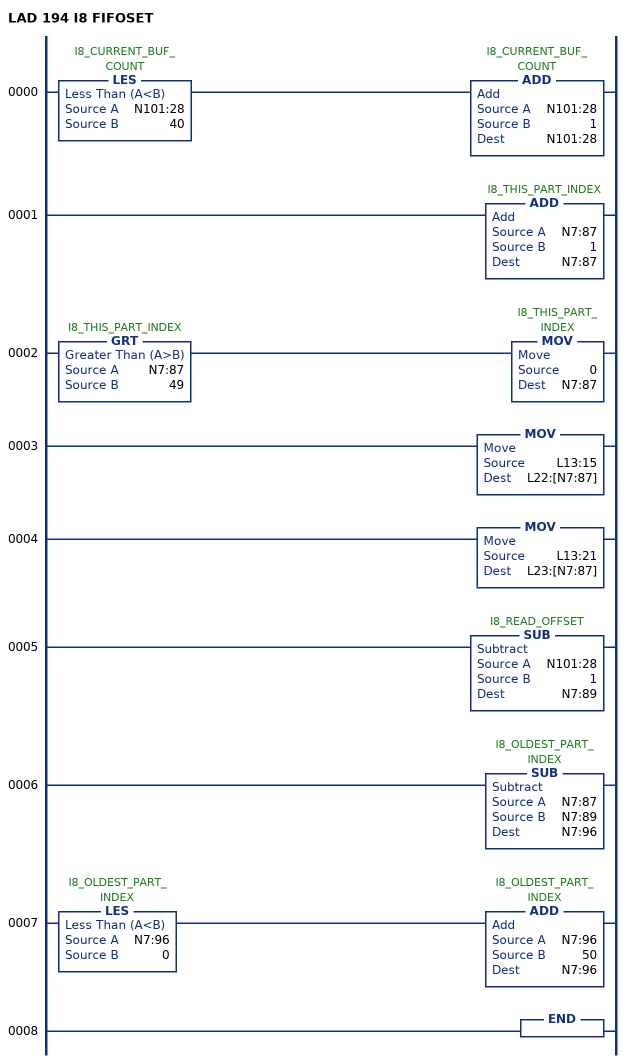
% Rung: 0 %
SOR LES N101:28 40 ADD N101:28 1 N101:28 EOR
%   N101:28  I8_CURRENT_BUF_COUNT %
% Rung: 1 %
SOR ADD N7:87 1 N7:87 EOR
%   N7:87  I8_THIS_PART_INDEX %
% Rung: 2 %
SOR GRT N7:87 49 MOV 0 N7:87 EOR
%   N7:87  I8_THIS_PART_INDEX %
% Rung: 3 %
SOR MOV L13:15 L22:[N7:87] EOR
%   L13:15  THE_TIME %
%   N7:87  I8_THIS_PART_INDEX %
% Rung: 4 %
SOR MOV L13:21 L23:[N7:87] EOR
%   L13:21  TOP_POSITION %
%   N7:87  I8_THIS_PART_INDEX %
% Rung: 5 %
SOR SUB N101:28 1 N7:89 EOR
%   N101:28  I8_CURRENT_BUF_COUNT %
%   N7:89  I8_READ_OFFSET %
% Rung: 6 %
SOR SUB N7:87 N7:89 N7:96 EOR
%   N7:87  I8_THIS_PART_INDEX %
%   N7:89  I8_READ_OFFSET %
%   N7:96  I8_OLDEST_PART_INDEX %
% Rung: 7 %
SOR LES N7:96 0 ADD N7:96 50 N7:96 EOR
%   N7:96  I8_OLDEST_PART_INDEX %
% Rung: 8 %
SOR END EOR

LADDER 195 "I8 FIFOGET"
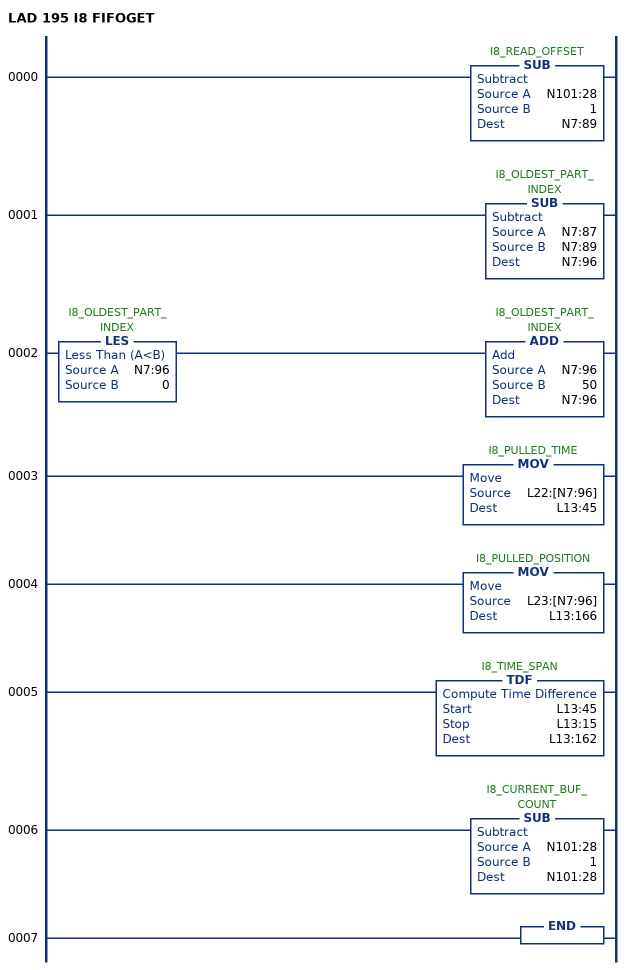
% Rung: 0 %
SOR SUB N101:28 1 N7:89 EOR
%   N101:28  I8_CURRENT_BUF_COUNT %
%   N7:89  I8_READ_OFFSET %
% Rung: 1 %
SOR SUB N7:87 N7:89 N7:96 EOR
%   N7:87  I8_THIS_PART_INDEX %
%   N7:89  I8_READ_OFFSET %
%   N7:96  I8_OLDEST_PART_INDEX %
% Rung: 2 %
SOR LES N7:96 0 ADD N7:96 50 N7:96 EOR
%   N7:96  I8_OLDEST_PART_INDEX %
% Rung: 3 %
SOR MOV L22:[N7:96] L13:45 EOR
%   N7:96  I8_OLDEST_PART_INDEX %
%   L13:45  I8_PULLED_TIME %
% Rung: 4 %
SOR MOV L23:[N7:96] L13:166 EOR
%   N7:96  I8_OLDEST_PART_INDEX %
%   L13:166  I8_PULLED_POSITION %
% Rung: 5 %
SOR TDF L13:45 L13:15 L13:162 EOR
%   L13:45  I8_PULLED_TIME %
%   L13:15  THE_TIME %
%   L13:162  I8_TIME_SPAN %
% Rung: 6 %
SOR SUB N101:28 1 N101:28 EOR
%   N101:28  I8_CURRENT_BUF_COUNT %
% Rung: 7 %
SOR END EOR

LADDER 196 "I8 DATA"
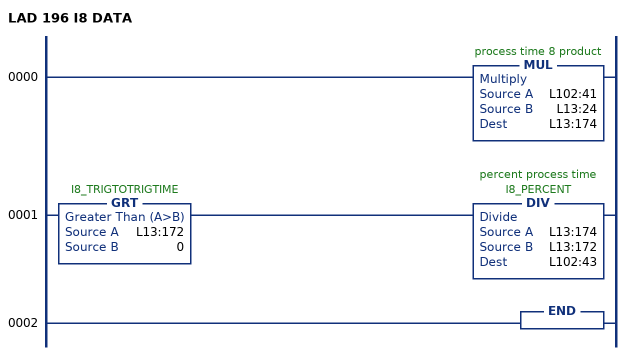
% Rung: 0 %
SOR MUL L102:41 L13:24 L13:174 EOR
%   L102:41  I8_PROCESSTIME %
%   L13:24  "multiplyer to make devision come out to a percentage" %
%   L13:174  "process time 8 product" %
% Rung: 1 %
SOR GRT L13:172 0 DIV L13:174 L13:172 L102:43 EOR
%   L13:172  I8_TRIGTOTRIGTIME %
%   L13:174  "process time 8 product" %
%   L102:43  I8_PERCENT  "percent process time" %
% Rung: 2 %
SOR END EOR

LADDER 197 "I8 FAULT"
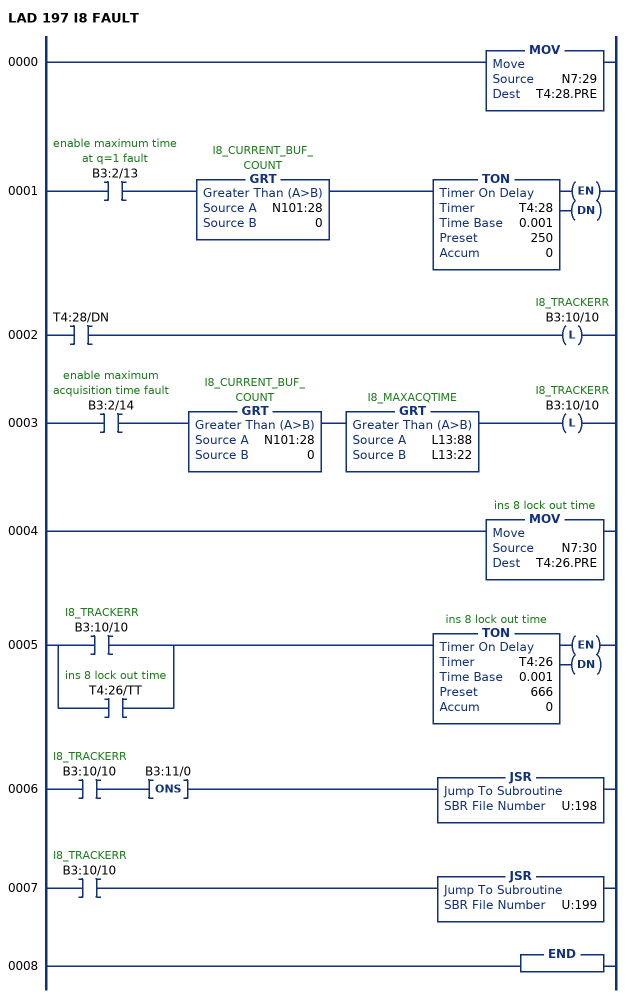
% Rung: 0 %
SOR MOV N7:29 T4:28.PRE EOR
%   N7:29  "max allowed ms time for q to be above 1 if safe fault is used" %
% Rung: 1 %
SOR XIC B3:2/13 GRT N101:28 0 TON T4:28 0.001 250 0 EOR
%   B3:2/13  "enable maximum time at q=1 fault" %
%   N101:28  I8_CURRENT_BUF_COUNT %
% Rung: 2 %
SOR XIC T4:28/DN OTL B3:10/10 EOR
%   B3:10/10  I8_TRACKERR %
% Rung: 3 %
SOR XIC B3:2/14 GRT N101:28 0 GRT L13:88 L13:22 OTL B3:10/10 EOR
%   B3:2/14  "enable maximum acquisition time fault" %
%   N101:28  I8_CURRENT_BUF_COUNT %
%   L13:88  I8_MAXACQTIME %
%   L13:22  "maximum of the longest acquire time allowed if maximum acquire time fault is enabled" %
%   B3:10/10  I8_TRACKERR %
% Rung: 4 %
SOR MOV N7:30 T4:26.PRE EOR
%   N7:30  "ms time setting to lock out inspection to give all pending images a chance to clear" %
%   T4:26  "ins 8 lock out time" %
% Rung: 5 %
SOR BST XIC B3:10/10 NXB XIC T4:26/TT BND TON T4:26 0.001 666 0 EOR
%   B3:10/10  I8_TRACKERR %
%   T4:26  "ins 8 lock out time" %
% Rung: 6 %
SOR XIC B3:10/10 ONS B3:11/0 JSR U:198 EOR
%   B3:10/10  I8_TRACKERR %
% Rung: 7 %
SOR XIC B3:10/10 JSR U:199 EOR
%   B3:10/10  I8_TRACKERR %
% Rung: 8 %
SOR END EOR

LADDER 198 "I8 FIX1"
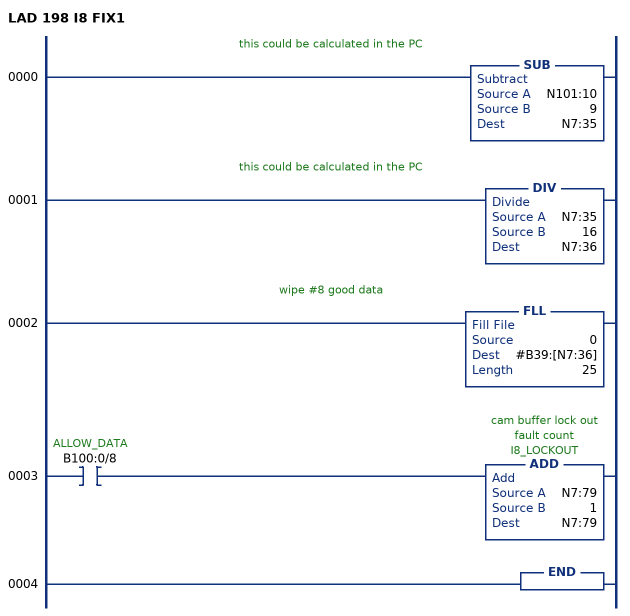
% Rung: 0 %
% this could be calculated in the PC %
SOR SUB N101:10 9 N7:35 EOR
%   N101:10  I8_TRIG_LOC %
% Rung: 1 %
% this could be calculated in the PC %
SOR DIV N7:35 16 N7:36 EOR
% Rung: 2 %
% wipe #8 good data %
SOR FLL 0 #B39:[N7:36] 25 EOR
% Rung: 3 %
SOR XIC B100:0/8 ADD N7:79 1 N7:79 EOR
%   B100:0/8  ALLOW_DATA %
%   N7:79  I8_LOCKOUT  "cam buffer lock out fault count" %
% Rung: 4 %
SOR END EOR

LADDER 199 "I8 FIX2"
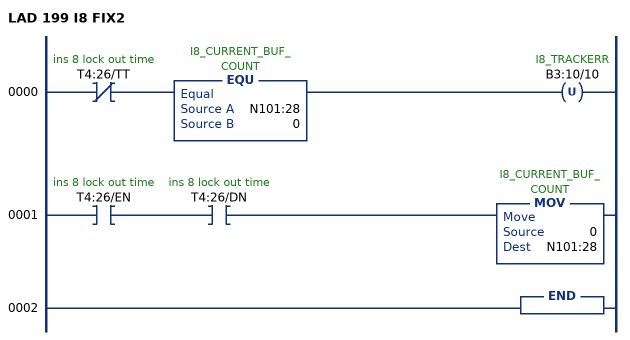
% Rung: 0 %
SOR XIO T4:26/TT EQU N101:28 0 OTU B3:10/10 EOR
%   T4:26  "ins 8 lock out time" %
%   N101:28  I8_CURRENT_BUF_COUNT %
%   B3:10/10  I8_TRACKERR %
% Rung: 1 %
SOR XIC T4:26/EN XIC T4:26/DN MOV 0 N101:28 EOR
%   T4:26  "ins 8 lock out time" %
%   N101:28  I8_CURRENT_BUF_COUNT %
% Rung: 2 %
SOR END EOR

LADDER 200 "PASS BLOW"
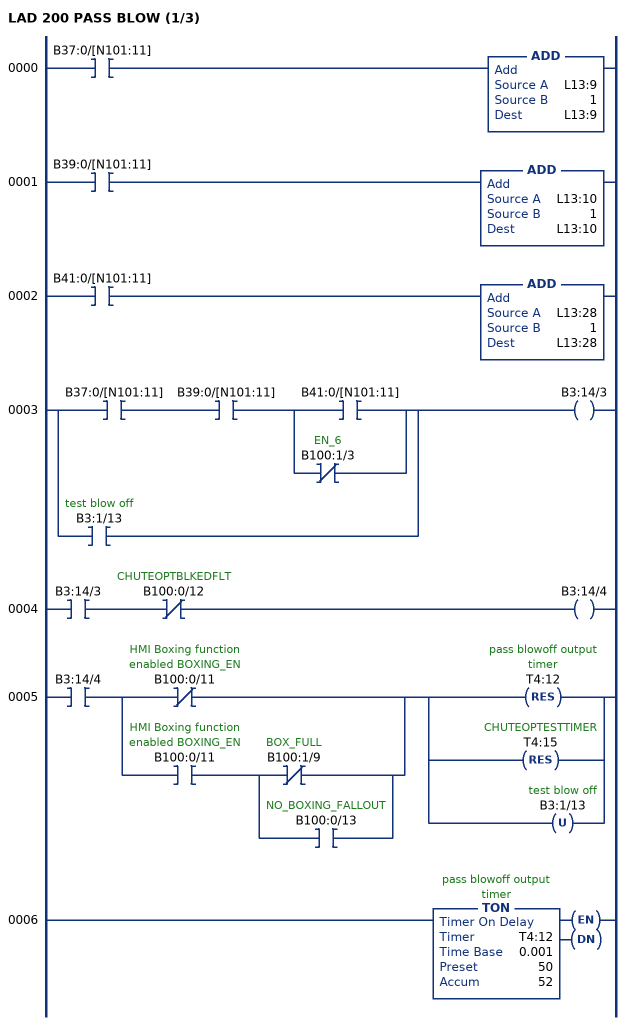
% Rung: 0 %
SOR XIC B37:0/[N101:11] ADD L13:9 1 L13:9 EOR
%   B37:0  TOP_OK_1 %
%   N101:11  BLOW_PT %
% Rung: 1 %
SOR XIC B39:0/[N101:11] ADD L13:10 1 L13:10 EOR
%   B39:0  TOP_OK_2 %
%   N101:11  BLOW_PT %
% Rung: 2 %
SOR XIC B41:0/[N101:11] ADD L13:28 1 L13:28 EOR
%   B41:0  TOP_OK_3 %
%   N101:11  BLOW_PT %
% Rung: 3 %
SOR BST XIC B37:0/[N101:11] XIC B39:0/[N101:11] BST XIC B41:0/[N101:11] NXB XIO B100:1/3 BND NXB XIC B3:1/13 BND OTE B3:14/3 EOR
%   B37:0  TOP_OK_1 %
%   N101:11  BLOW_PT %
%   B39:0  TOP_OK_2 %
%   B41:0  TOP_OK_3 %
%   B100:1/3  EN_6 %
%   B3:1/13  "test blow off" %
% Rung: 4 %
SOR XIC B3:14/3 XIO B100:0/12 OTE B3:14/4 EOR
%   B100:0/12  CHUTEOPTBLKEDFLT %
% Rung: 5 %
SOR XIC B3:14/4 BST XIO B100:0/11 NXB XIC B100:0/11 BST XIO B100:1/9 NXB XIC B100:0/13 BND BND BST RES T4:12 NXB RES T4:15 NXB OTU B3:1/13 BND EOR
%   B100:0/11  BOXING_EN  "HMI Boxing function enabled" %
%   B100:1/9  BOX_FULL %
%   B100:0/13  NO_BOXING_FALLOUT %
%   T4:12  "pass blowoff output timer" %
%   T4:15  CHUTEOPTESTTIMER %
%   B3:1/13  "test blow off" %
% Rung: 6 %
SOR TON T4:12 0.001 50 52 EOR
%   T4:12  "pass blowoff output timer" %

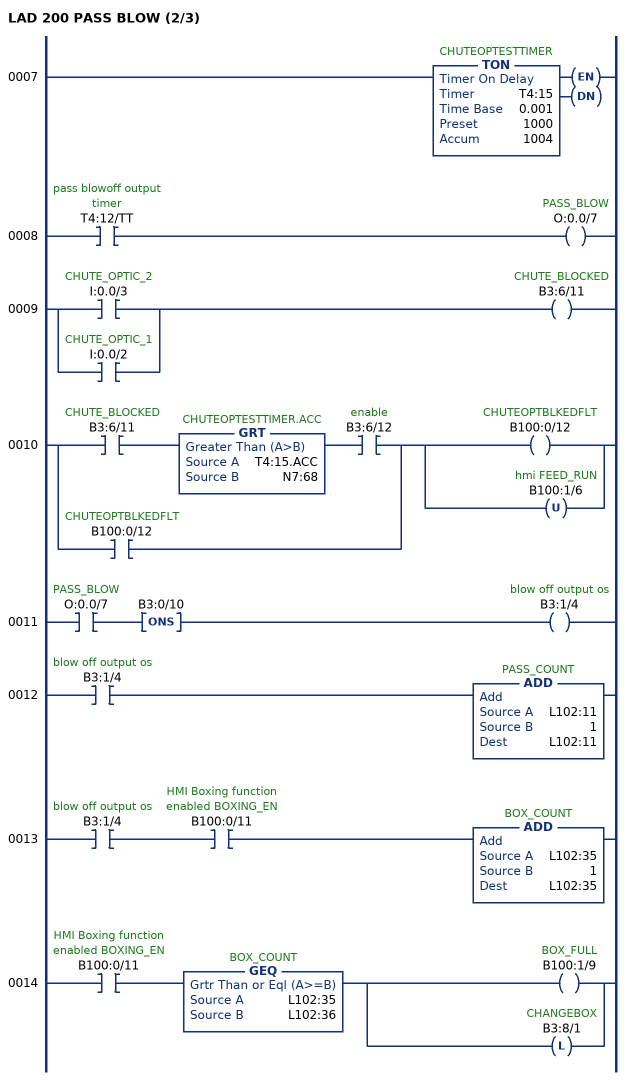
% Rung: 7 %
SOR TON T4:15 0.001 1000 1004 EOR
%   T4:15  CHUTEOPTESTTIMER %
% Rung: 8 %
SOR XIC T4:12/TT OTE O:0.0/7 EOR
%   T4:12  "pass blowoff output timer" %
%   O:0.0/7  PASS_BLOW %
% Rung: 9 %
SOR BST XIC I:0.0/3 NXB XIC I:0.0/2 BND OTE B3:6/11 EOR
%   I:0.0/3  CHUTE_OPTIC_2 %
%   I:0.0/2  CHUTE_OPTIC_1 %
%   B3:6/11  CHUTE_BLOCKED %
% Rung: 10 %
SOR BST XIC B3:6/11 GRT T4:15.ACC N7:68 XIC B3:6/12 NXB XIC B100:0/12 BND BST OTE B100:0/12 NXB OTU B100:1/6 BND EOR
%   B3:6/11  CHUTE_BLOCKED %
%   T4:15  CHUTEOPTESTTIMER %
%   B3:6/12  "enable" %
%   B100:0/12  CHUTEOPTBLKEDFLT %
%   B100:1/6  FEED_RUN  "hmi" %
% Rung: 11 %
SOR XIC O:0.0/7 ONS B3:0/10 OTE B3:1/4 EOR
%   O:0.0/7  PASS_BLOW %
%   B3:1/4  "blow off output os" %
% Rung: 12 %
SOR XIC B3:1/4 ADD L102:11 1 L102:11 EOR
%   B3:1/4  "blow off output os" %
%   L102:11  PASS_COUNT %
% Rung: 13 %
SOR XIC B3:1/4 XIC B100:0/11 ADD L102:35 1 L102:35 EOR
%   B3:1/4  "blow off output os" %
%   B100:0/11  BOXING_EN  "HMI Boxing function enabled" %
%   L102:35  BOX_COUNT %
% Rung: 14 %
SOR XIC B100:0/11 GEQ L102:35 L102:36 BST OTE B100:1/9 NXB OTL B3:8/1 BND EOR
%   B100:0/11  BOXING_EN  "HMI Boxing function enabled" %
%   L102:35  BOX_COUNT %
%   L102:36  BOX_LIMIT  "box count setpoint" %
%   B100:1/9  BOX_FULL %
%   B3:8/1  CHANGEBOX %

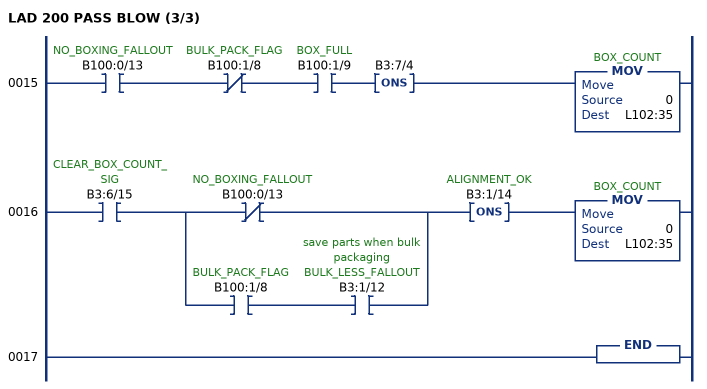
% Rung: 15 %
SOR XIC B100:0/13 XIO B100:1/8 XIC B100:1/9 ONS B3:7/4 MOV 0 L102:35 EOR
%   B100:0/13  NO_BOXING_FALLOUT %
%   B100:1/8  BULK_PACK_FLAG %
%   B100:1/9  BOX_FULL %
%   L102:35  BOX_COUNT %
% Rung: 16 %
SOR XIC B3:6/15 BST XIO B100:0/13 NXB XIC B100:1/8 XIC B3:1/12 BND ONS B3:1/14 MOV 0 L102:35 EOR
%   B3:6/15  CLEAR_BOX_COUNT_SIG %
%   B100:0/13  NO_BOXING_FALLOUT %
%   B100:1/8  BULK_PACK_FLAG %
%   B3:1/12  BULK_LESS_FALLOUT  "save parts when bulk packaging" %
%   B3:1/14  ALIGNMENT_OK %
%   L102:35  BOX_COUNT %
% Rung: 17 %
SOR END EOR

LADDER 235 "TESTTRIGS"    % highspeed test triggers, not necessary %
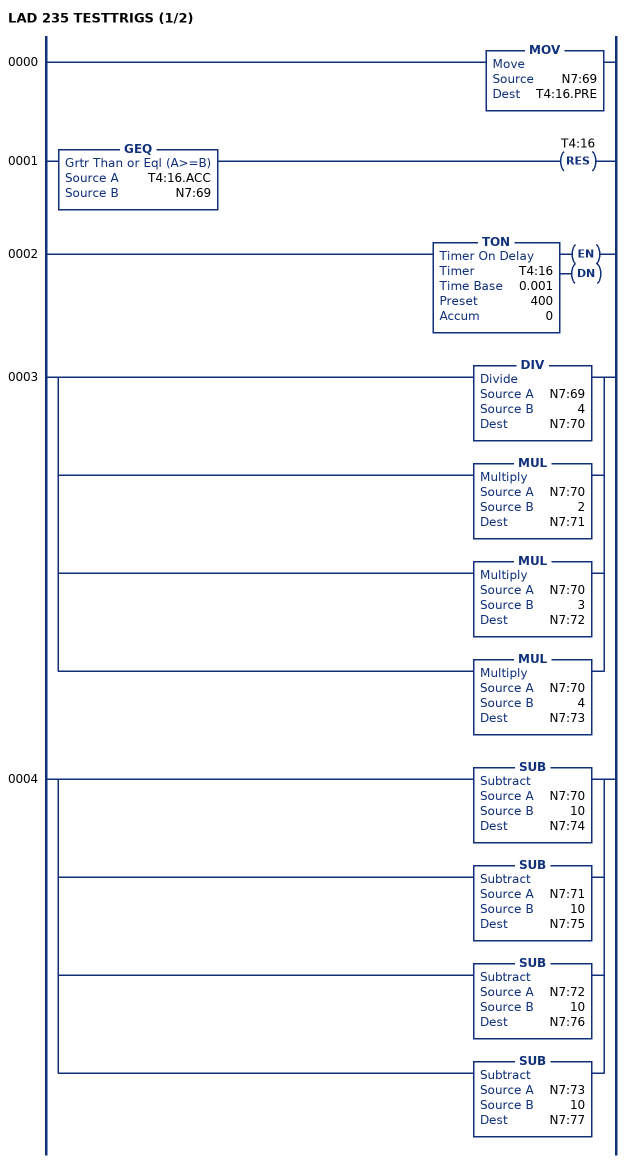
% Rung: 0 %
SOR MOV N7:69 T4:16.PRE EOR
% Rung: 1 %
SOR GEQ T4:16.ACC N7:69 RES T4:16 EOR
% Rung: 2 %
SOR TON T4:16 0.001 400 0 EOR
% Rung: 3 %
SOR BST DIV N7:69 4 N7:70 NXB MUL N7:70 2 N7:71 NXB MUL N7:70 3 N7:72 NXB MUL N7:70 4 N7:73 BND EOR
% Rung: 4 %
SOR BST SUB N7:70 10 N7:74 NXB SUB N7:71 10 N7:75 NXB SUB N7:72 10 N7:76 NXB SUB N7:73 10 N7:77 BND EOR

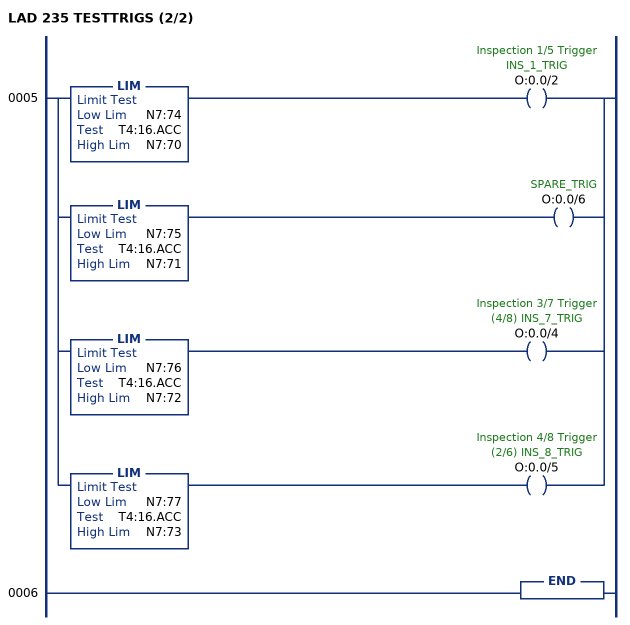
% Rung: 5 %
SOR BST LIM N7:74 T4:16.ACC N7:70 OTE O:0.0/2 NXB LIM N7:75 T4:16.ACC N7:71 OTE O:0.0/6 NXB LIM N7:76 T4:16.ACC N7:72 OTE O:0.0/4 NXB LIM N7:77 T4:16.ACC N7:73 OTE O:0.0/5 BND EOR
%   O:0.0/2  INS_1_TRIG  "Inspection 1/5 Trigger" %
%   O:0.0/6  SPARE_TRIG %
%   O:0.0/4  INS_7_TRIG  "Inspection 3/7 Trigger (4/8)" %
%   O:0.0/5  INS_8_TRIG  "Inspection 4/8 Trigger (2/6)" %
% Rung: 6 %
SOR END EOR

LADDER 236 "TESTTRIG1"
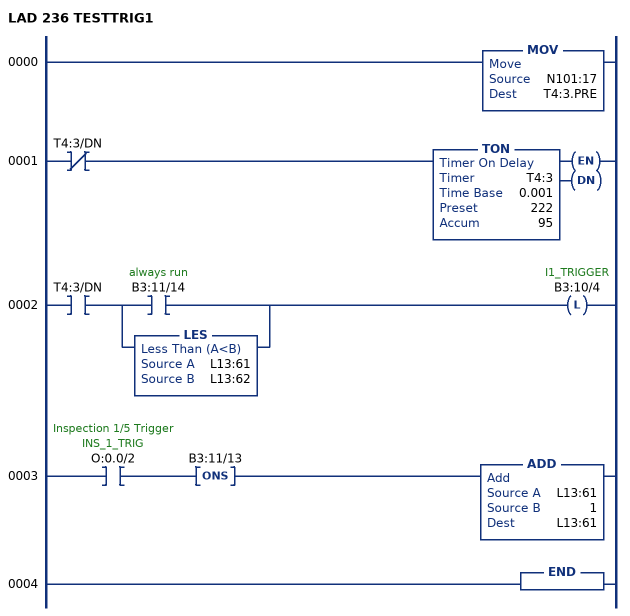
% Rung: 0 %
SOR MOV N101:17 T4:3.PRE EOR
%   N101:17  I1_TRIGTIME  "test trigger 1 interval" %
% Rung: 1 %
SOR XIO T4:3/DN TON T4:3 0.001 222 95 EOR
% Rung: 2 %
SOR XIC T4:3/DN BST XIC B3:11/14 NXB LES L13:61 L13:62 BND OTL B3:10/4 EOR
%   B3:11/14  "always run" %
%   B3:10/4  I1_TRIGGER %
% Rung: 3 %
SOR XIC O:0.0/2 ONS B3:11/13 ADD L13:61 1 L13:61 EOR
%   O:0.0/2  INS_1_TRIG  "Inspection 1/5 Trigger" %
% Rung: 4 %
SOR END EOR

LADDER 237 "TESTTRIG2"
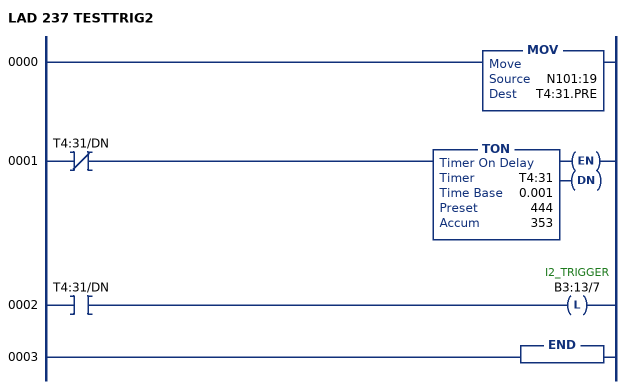
% Rung: 0 %
SOR MOV N101:19 T4:31.PRE EOR
%   N101:19  I2_I6_TRIGTIME  "test trgiger 2/6 interval" %
% Rung: 1 %
SOR XIO T4:31/DN TON T4:31 0.001 444 353 EOR
% Rung: 2 %
SOR XIC T4:31/DN OTL B3:13/7 EOR
%   B3:13/7  I2_TRIGGER %
% Rung: 3 %
SOR END EOR

LADDER 238 "TESTTRIG3"
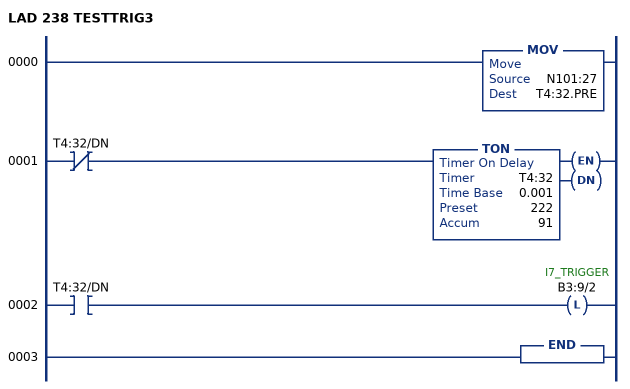
% Rung: 0 %
SOR MOV N101:27 T4:32.PRE EOR
%   N101:27  I7_TRIGTIME %
% Rung: 1 %
SOR XIO T4:32/DN TON T4:32 0.001 222 91 EOR
% Rung: 2 %
SOR XIC T4:32/DN OTL B3:9/2 EOR
%   B3:9/2  I7_TRIGGER %
% Rung: 3 %
SOR END EOR

LADDER 239 "TESTTRIG4"
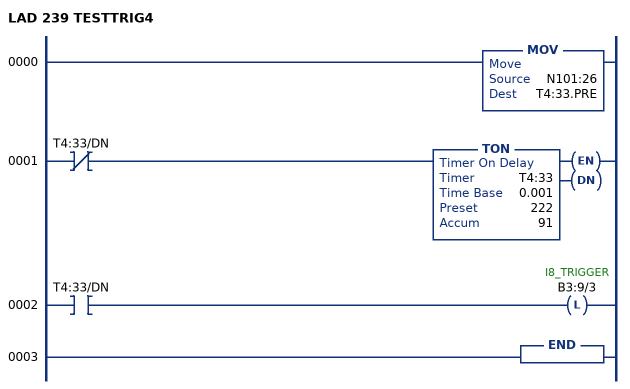
% Rung: 0 %
SOR MOV N101:26 T4:33.PRE EOR
%   N101:26  I8_TRIGTIME %
% Rung: 1 %
SOR XIO T4:33/DN TON T4:33 0.001 222 91 EOR
% Rung: 2 %
SOR XIC T4:33/DN OTL B3:9/3 EOR
%   B3:9/3  I8_TRIGGER %
% Rung: 3 %
SOR END EOR

LADDER 240 "TESTTRIG5"
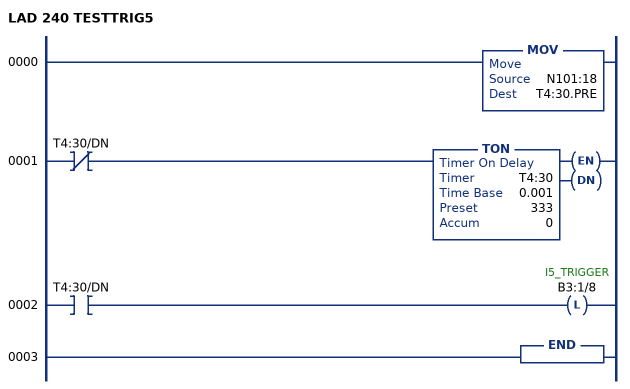
% Rung: 0 %
SOR MOV N101:18 T4:30.PRE EOR
%   N101:18  I5_TRIGTIME  "test trigger 5 interval" %
% Rung: 1 %
SOR XIO T4:30/DN TON T4:30 0.001 333 0 EOR
% Rung: 2 %
SOR XIC T4:30/DN OTL B3:1/8 EOR
%   B3:1/8  I5_TRIGGER %
% Rung: 3 %
SOR END EOR

LADDER 241 "TESTTRIG6"
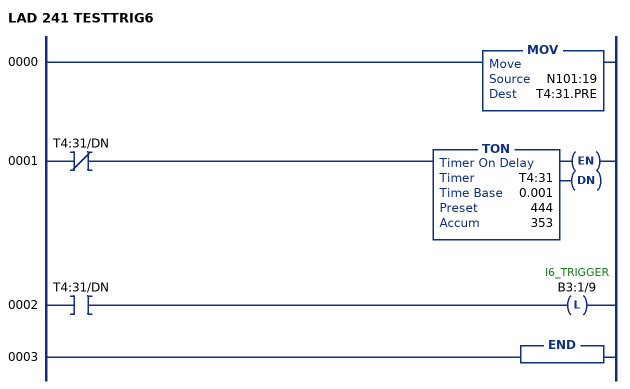
% Rung: 0 %
SOR MOV N101:19 T4:31.PRE EOR
%   N101:19  I2_I6_TRIGTIME  "test trgiger 2/6 interval" %
% Rung: 1 %
SOR XIO T4:31/DN TON T4:31 0.001 444 353 EOR
% Rung: 2 %
SOR XIC T4:31/DN OTL B3:1/9 EOR
%   B3:1/9  I6_TRIGGER %
% Rung: 3 %
SOR END EOR

LADDER 242 "TESTTRIG7"
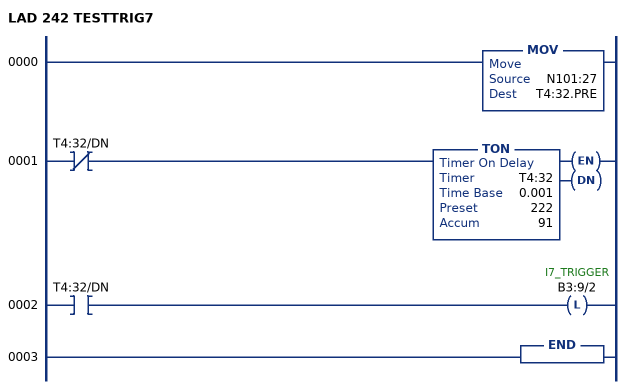
% Rung: 0 %
SOR MOV N101:27 T4:32.PRE EOR
%   N101:27  I7_TRIGTIME %
% Rung: 1 %
SOR XIO T4:32/DN TON T4:32 0.001 222 91 EOR
% Rung: 2 %
SOR XIC T4:32/DN OTL B3:9/2 EOR
%   B3:9/2  I7_TRIGGER %
% Rung: 3 %
SOR END EOR

LADDER 243 "TESTTRIG8"
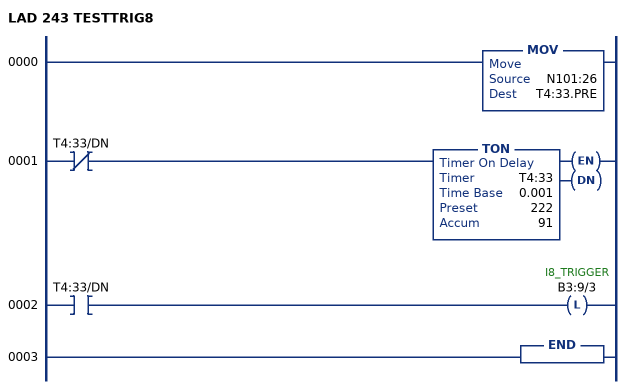
% Rung: 0 %
SOR MOV N101:26 T4:33.PRE EOR
%   N101:26  I8_TRIGTIME %
% Rung: 1 %
SOR XIO T4:33/DN TON T4:33 0.001 222 91 EOR
% Rung: 2 %
SOR XIC T4:33/DN OTL B3:9/3 EOR
%   B3:9/3  I8_TRIGGER %
% Rung: 3 %
SOR END EOR

LADDER 244 "PACKAGER"    % normal %
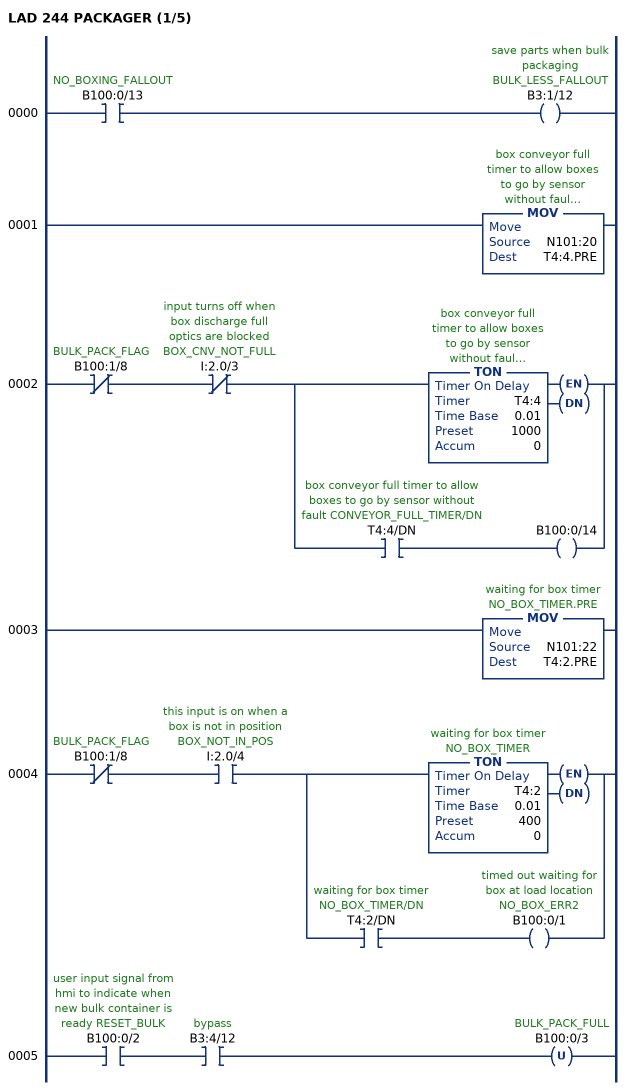
% Rung: 0 %
SOR XIC B100:0/13 OTE B3:1/12 EOR
%   B100:0/13  NO_BOXING_FALLOUT %
%   B3:1/12  BULK_LESS_FALLOUT  "save parts when bulk packaging" %
% Rung: 1 %
SOR MOV N101:20 T4:4.PRE EOR
%   N101:20  CONV_FULL_TIME_LIMIT  "time to allow box to pass box conveyor full sensor without fault" %
%   T4:4  CONVEYOR_FULL_TIMER  "box conveyor full timer to allow boxes to go by sensor without fault" %
% Rung: 2 %
SOR XIO B100:1/8 XIO I:2.0/3 BST TON T4:4 0.01 1000 0 NXB XIC T4:4/DN OTE B100:0/14 BND EOR
%   B100:1/8  BULK_PACK_FLAG %
%   I:2.0/3  BOX_CNV_NOT_FULL  "input turns off when box discharge full optics are blocked" %
%   T4:4  CONVEYOR_FULL_TIMER  "box conveyor full timer to allow boxes to go by sensor without fault" %
% Rung: 3 %
SOR MOV N101:22 T4:2.PRE EOR
%   N101:22  BOX_WAIT_TIME_LIMIT  "the time until waiting for box message in hmi (fault)" %
%   T4:2  NO_BOX_TIMER  "waiting for box timer" %
% Rung: 4 %
SOR XIO B100:1/8 XIC I:2.0/4 BST TON T4:2 0.01 400 0 NXB XIC T4:2/DN OTE B100:0/1 BND EOR
%   B100:1/8  BULK_PACK_FLAG %
%   I:2.0/4  BOX_NOT_IN_POS  "this input is on when a box is not in position" %
%   T4:2  NO_BOX_TIMER  "waiting for box timer" %
%   B100:0/1  NO_BOX_ERR2  "timed out waiting for box at load location" %
% Rung: 5 %
SOR XIC B100:0/2 XIC B3:4/12 OTU B100:0/3 EOR
%   B100:0/2  RESET_BULK  "user input signal from hmi to indicate when new bulk container is ready" %
%   B3:4/12  "bypass" %
%   B100:0/3  BULK_PACK_FULL %

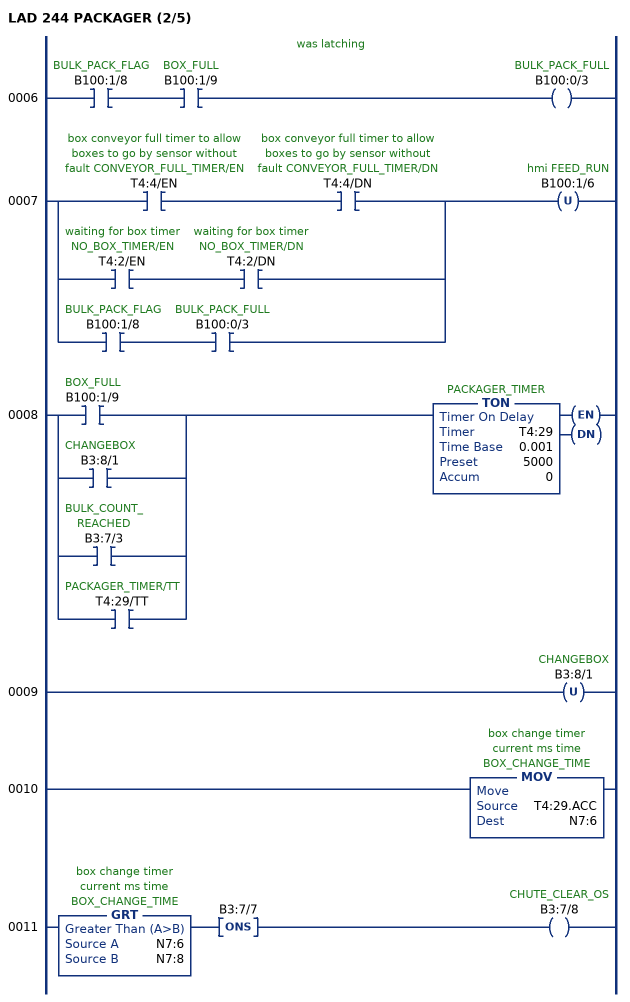
% Rung: 6 %
% was latching %
SOR XIC B100:1/8 XIC B100:1/9 OTE B100:0/3 EOR
%   B100:1/8  BULK_PACK_FLAG %
%   B100:1/9  BOX_FULL %
%   B100:0/3  BULK_PACK_FULL %
% Rung: 7 %
SOR BST XIC T4:4/EN XIC T4:4/DN NXB XIC T4:2/EN XIC T4:2/DN NXB XIC B100:1/8 XIC B100:0/3 BND OTU B100:1/6 EOR
%   T4:4  CONVEYOR_FULL_TIMER  "box conveyor full timer to allow boxes to go by sensor without fault" %
%   T4:2  NO_BOX_TIMER  "waiting for box timer" %
%   B100:1/8  BULK_PACK_FLAG %
%   B100:0/3  BULK_PACK_FULL %
%   B100:1/6  FEED_RUN  "hmi" %
% Rung: 8 %
SOR BST XIC B100:1/9 NXB XIC B3:8/1 NXB XIC B3:7/3 NXB XIC T4:29/TT BND TON T4:29 0.001 5000 0 EOR
%   B100:1/9  BOX_FULL %
%   B3:8/1  CHANGEBOX %
%   B3:7/3  BULK_COUNT_REACHED %
%   T4:29  PACKAGER_TIMER %
% Rung: 9 %
SOR OTU B3:8/1 EOR
%   B3:8/1  CHANGEBOX %
% Rung: 10 %
SOR MOV T4:29.ACC N7:6 EOR
%   T4:29  PACKAGER_TIMER %
%   N7:6  BOX_CHANGE_TIME  "box change timer current ms time" %
% Rung: 11 %
SOR GRT N7:6 N7:8 ONS B3:7/7 OTE B3:7/8 EOR
%   N7:6  BOX_CHANGE_TIME  "box change timer current ms time" %
%   N7:8  CHUTE_CLEAR_TIME %
%   B3:7/8  CHUTE_CLEAR_OS %

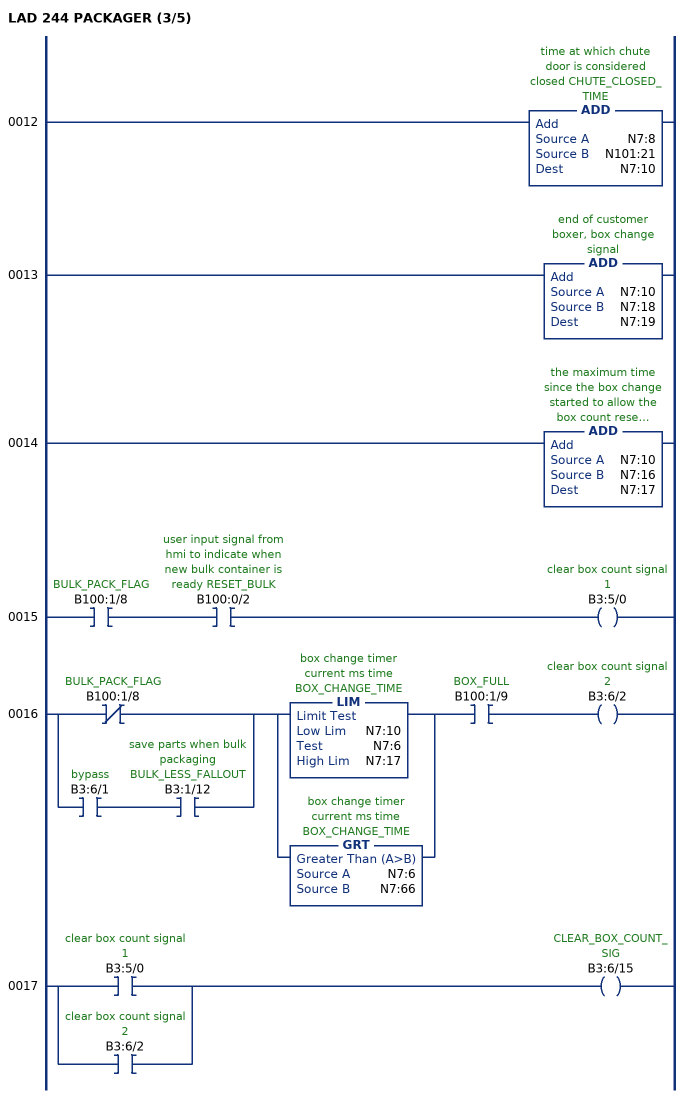
% Rung: 12 %
SOR ADD N7:8 N101:21 N7:10 EOR
%   N7:8  CHUTE_CLEAR_TIME %
%   N101:21  CHUTE_CLOSE_TIME  "ms time required to close chute" %
%   N7:10  CHUTE_CLOSED_TIME  "time at which chute door is considered closed" %
% Rung: 13 %
SOR ADD N7:10 N7:18 N7:19 EOR
%   N7:10  CHUTE_CLOSED_TIME  "time at which chute door is considered closed" %
%   N7:18  CHANGE_BOX_SIG_TIME  "customer boxer change box signal time" %
%   N7:19  "end of customer boxer, box change signal" %
% Rung: 14 %
SOR ADD N7:10 N7:16 N7:17 EOR
%   N7:10  CHUTE_CLOSED_TIME  "time at which chute door is considered closed" %
%   N7:16  RESET_COUNT_SIG_TIME  "maximum length of time to hold box count reset signal on" %
%   N7:17  "the maximum time since the box change started to allow the box count reset signal" %
% Rung: 15 %
SOR XIC B100:1/8 XIC B100:0/2 OTE B3:5/0 EOR
%   B100:1/8  BULK_PACK_FLAG %
%   B100:0/2  RESET_BULK  "user input signal from hmi to indicate when new bulk container is ready" %
%   B3:5/0  "clear box count signal 1" %
% Rung: 16 %
SOR BST XIO B100:1/8 NXB XIC B3:6/1 XIC B3:1/12 BND BST LIM N7:10 N7:6 N7:17 NXB GRT N7:6 N7:66 BND XIC B100:1/9 OTE B3:6/2 EOR
%   B100:1/8  BULK_PACK_FLAG %
%   B3:6/1  "bypass" %
%   B3:1/12  BULK_LESS_FALLOUT  "save parts when bulk packaging" %
%   N7:10  CHUTE_CLOSED_TIME  "time at which chute door is considered closed" %
%   N7:6  BOX_CHANGE_TIME  "box change timer current ms time" %
%   N7:17  "the maximum time since the box change started to allow the box count reset signal" %
%   B100:1/9  BOX_FULL %
%   B3:6/2  "clear box count signal 2" %
% Rung: 17 %
SOR BST XIC B3:5/0 NXB XIC B3:6/2 BND OTE B3:6/15 EOR
%   B3:5/0  "clear box count signal 1" %
%   B3:6/2  "clear box count signal 2" %
%   B3:6/15  CLEAR_BOX_COUNT_SIG %

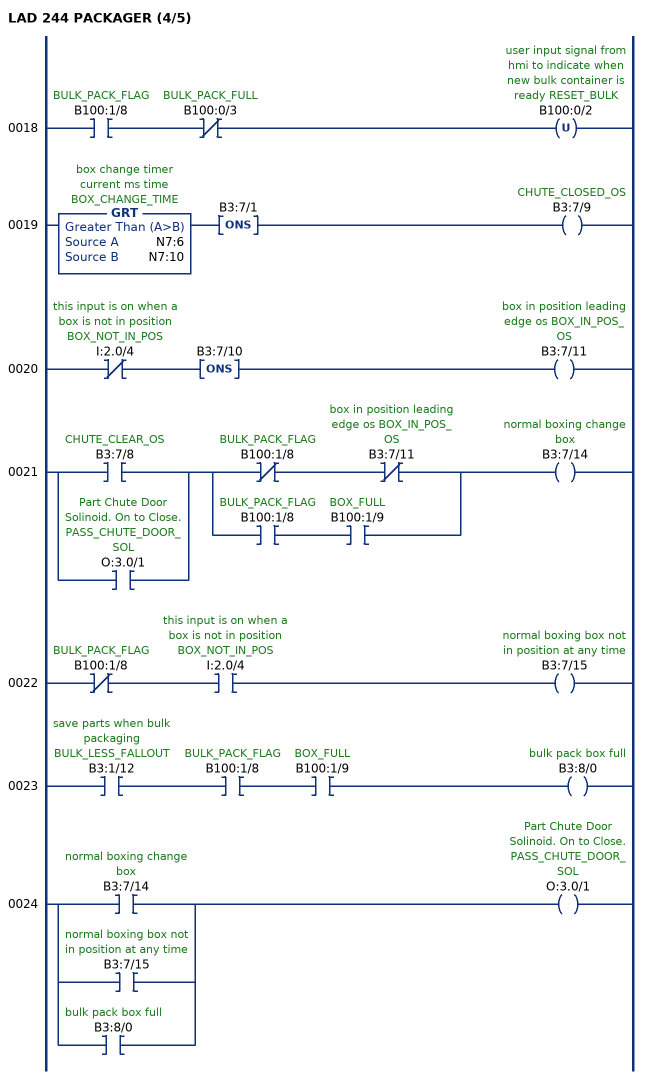
% Rung: 18 %
SOR XIC B100:1/8 XIO B100:0/3 OTU B100:0/2 EOR
%   B100:1/8  BULK_PACK_FLAG %
%   B100:0/3  BULK_PACK_FULL %
%   B100:0/2  RESET_BULK  "user input signal from hmi to indicate when new bulk container is ready" %
% Rung: 19 %
SOR GRT N7:6 N7:10 ONS B3:7/1 OTE B3:7/9 EOR
%   N7:6  BOX_CHANGE_TIME  "box change timer current ms time" %
%   N7:10  CHUTE_CLOSED_TIME  "time at which chute door is considered closed" %
%   B3:7/9  CHUTE_CLOSED_OS %
% Rung: 20 %
SOR XIO I:2.0/4 ONS B3:7/10 OTE B3:7/11 EOR
%   I:2.0/4  BOX_NOT_IN_POS  "this input is on when a box is not in position" %
%   B3:7/11  BOX_IN_POS_OS  "box in position leading edge os" %
% Rung: 21 %
SOR BST XIC B3:7/8 NXB XIC O:3.0/1 BND BST XIO B100:1/8 XIO B3:7/11 NXB XIC B100:1/8 XIC B100:1/9 BND OTE B3:7/14 EOR
%   B3:7/8  CHUTE_CLEAR_OS %
%   O:3.0/1  PASS_CHUTE_DOOR_SOL  "Part Chute Door Solinoid. On to Close." %
%   B100:1/8  BULK_PACK_FLAG %
%   B3:7/11  BOX_IN_POS_OS  "box in position leading edge os" %
%   B100:1/9  BOX_FULL %
%   B3:7/14  "normal boxing change box" %
% Rung: 22 %
SOR XIO B100:1/8 XIC I:2.0/4 OTE B3:7/15 EOR
%   B100:1/8  BULK_PACK_FLAG %
%   I:2.0/4  BOX_NOT_IN_POS  "this input is on when a box is not in position" %
%   B3:7/15  "normal boxing box not in position at any time" %
% Rung: 23 %
SOR XIC B3:1/12 XIC B100:1/8 XIC B100:1/9 OTE B3:8/0 EOR
%   B3:1/12  BULK_LESS_FALLOUT  "save parts when bulk packaging" %
%   B100:1/8  BULK_PACK_FLAG %
%   B100:1/9  BOX_FULL %
%   B3:8/0  "bulk pack box full" %
% Rung: 24 %
SOR BST XIC B3:7/14 NXB XIC B3:7/15 NXB XIC B3:8/0 BND OTE O:3.0/1 EOR
%   B3:7/14  "normal boxing change box" %
%   B3:7/15  "normal boxing box not in position at any time" %
%   B3:8/0  "bulk pack box full" %
%   O:3.0/1  PASS_CHUTE_DOOR_SOL  "Part Chute Door Solinoid. On to Close." %

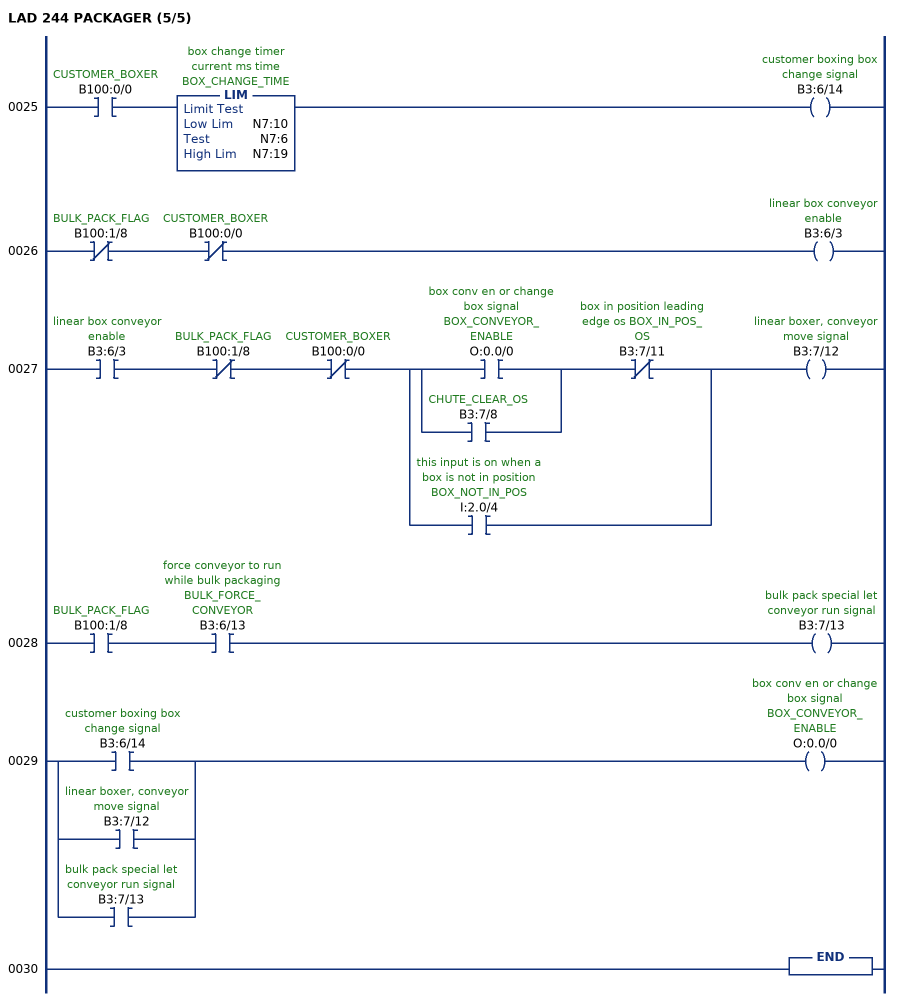
% Rung: 25 %
SOR XIC B100:0/0 LIM N7:10 N7:6 N7:19 OTE B3:6/14 EOR
%   B100:0/0  CUSTOMER_BOXER %
%   N7:10  CHUTE_CLOSED_TIME  "time at which chute door is considered closed" %
%   N7:6  BOX_CHANGE_TIME  "box change timer current ms time" %
%   N7:19  "end of customer boxer, box change signal" %
%   B3:6/14  "customer boxing box change signal" %
% Rung: 26 %
SOR XIO B100:1/8 XIO B100:0/0 OTE B3:6/3 EOR
%   B100:1/8  BULK_PACK_FLAG %
%   B100:0/0  CUSTOMER_BOXER %
%   B3:6/3  "linear box conveyor enable" %
% Rung: 27 %
SOR XIC B3:6/3 XIO B100:1/8 XIO B100:0/0 BST BST XIC O:0.0/0 NXB XIC B3:7/8 BND XIO B3:7/11 NXB XIC I:2.0/4 BND OTE B3:7/12 EOR
%   B3:6/3  "linear box conveyor enable" %
%   B100:1/8  BULK_PACK_FLAG %
%   B100:0/0  CUSTOMER_BOXER %
%   O:0.0/0  BOX_CONVEYOR_ENABLE  "box conv en or change box signal" %
%   B3:7/8  CHUTE_CLEAR_OS %
%   B3:7/11  BOX_IN_POS_OS  "box in position leading edge os" %
%   I:2.0/4  BOX_NOT_IN_POS  "this input is on when a box is not in position" %
%   B3:7/12  "linear boxer, conveyor move signal" %
% Rung: 28 %
SOR XIC B100:1/8 XIC B3:6/13 OTE B3:7/13 EOR
%   B100:1/8  BULK_PACK_FLAG %
%   B3:6/13  BULK_FORCE_CONVEYOR  "force conveyor to run while bulk packaging" %
%   B3:7/13  "bulk pack special let conveyor run signal" %
% Rung: 29 %
SOR BST XIC B3:6/14 NXB XIC B3:7/12 NXB XIC B3:7/13 BND OTE O:0.0/0 EOR
%   B3:6/14  "customer boxing box change signal" %
%   B3:7/12  "linear boxer, conveyor move signal" %
%   B3:7/13  "bulk pack special let conveyor run signal" %
%   O:0.0/0  BOX_CONVEYOR_ENABLE  "box conv en or change box signal" %
% Rung: 30 %
SOR END EOR

LADDER 245 "NO PACKAGE"
